{attribute 'GeneratedUsingTerminal: EL3314-0000-0016'}
{attribute addProperty BoxType "EL3314-0000-0016"}
{attribute addProperty Description "EL3314 4Ch. Ana. Input Thermocouple (TC)"}
{attribute addProperty Physics "KK"}
{attribute addProperty Id "TC_Inputs_Channel_1AT %I*TC_Inputs_Channel_EA9DF21E9TC_Inputs_Channel_2AT %I*TC_Inputs_Channel_EA9DF21E9TC_Inputs_Channel_3AT %I*TC_Inputs_Channel_EA9DF21E9TC_Inputs_Channel_4AT %I*TC_Inputs_Channel_EA9DF21E9WcStateAT %I*WcState_9091E0EB2InfoDataAT %I*InfoData_32EB74EA10"}
{attribute addProperty CRC "414953287"}
{attribute addProperty Size "48"}
TYPE EL3314_18BBAF47 EXTENDS EtcSlaveTerminalBase_947E5A46 :
STRUCT
	{attribute addProperty Name "TC_Inputs_Channel_1"}
	TC_Inputs_Channel_1 : TC_Inputs_Channel_EA9DF21E;
	{attribute addProperty Name "TC_Inputs_Channel_2"}
	TC_Inputs_Channel_2 : TC_Inputs_Channel_EA9DF21E;
	{attribute addProperty Name "TC_Inputs_Channel_3"}
	TC_Inputs_Channel_3 : TC_Inputs_Channel_EA9DF21E;
	{attribute addProperty Name "TC_Inputs_Channel_4"}
	TC_Inputs_Channel_4 : TC_Inputs_Channel_EA9DF21E;
	{attribute addProperty Name "WcState"}
	WcState : WcState_9091E0EB;
	{attribute addProperty Name "InfoData"}
	InfoData : InfoData_32EB74EA;
END_STRUCT
END_TYPE

(* stored: Version 1.2.0.0, ProductVersion 3.1.4024.11
   DUT EL3314_18BBAF47: Id {85127fbd-1555-4359-ad51-0245271f5ea5} *)
